PROGRAM MAIN
VAR
	fbConveyor	: FB_Conveyor;
	sMode		: STRING;
END_VAR

fbConveyor(
	eModeCommand			:= , 
	eCommand				:= , 
	eMode					=> , 
	eState					=> , 
	bUndefinedDone			=> , 
	bInvalidModeCommandOut	=> , 
	bChangeIntoProduction	=> );
sMode := F_UnitModeToString(fbConveyor.eMode);

END_PROGRAM

(* stored: Version 1.1.0.1, ProductVersion 3.1.4024.10
   POU MAIN: Id {52398f7a-babb-4f85-9ef7-be3bd41343dc}, SpecialFunc None *)
